// TIA Portal V19 export
FUNCTION "STD_STEP_CONTROL_HEAT" : Void   // FC6, STL
TITLE = Step controller - Heater
{ S7_Optimized_Access := 'TRUE' }
AUTHOR : JOM
FAMILY : STD
NAME : REG0391
VERSION : 0.0
// Comment
// stored: AutoNumber false
   VAR_IN_OUT
      MANUEL : Bool;   // Controller in manuel mode
      AUTO : Bool;   // Controller in auto mode
      PV : Real;   // Process Variabel
      SP : Real;   // Set Point
      MAX_DELTA : Real;
      MIN_DELTA : Real;
      FAKTOR_LARGE : Int;
      FAKTOR_SMALL : Int;
      ANA_OUTPUT : Int;
   END_VAR
BEGIN

NETWORK
TITLE = Step controller - Heater
// Comment
      A     #MANUEL;
      JC    M001;  // MANUAL
      A     #AUTO;
      JC    M002;  // AUTOMATIC
      L     0;  // = 4,00 mA
      T     #ANA_OUTPUT;  // OUTPUT
      BEU;  // END
M002: NOP   0;
      L     #PV;  // MEASURED
      L     #SP;  // SETPOINT
      -R;
      L     #MAX_DELTA;  // MAX. DELTA
      >R;
      JC    M004;
      L     #SP;  // SETPOINT
      L     #PV;  // MEASURED
      -R;
      L     #MAX_DELTA;  // MAX. DELTA
      >R;
      JC    M003;
      L     #PV;  // MEASURED
      L     #SP;  // SETPOINT
      -R;
      L     #MIN_DELTA;  // MIN. DELTA
      >R;
      JC    M006;
      L     #SP;  // SETPOINT
      L     #PV;  // MEASURED
      -R;
      L     #MIN_DELTA;  // MIN. DELTA
      >R;
      JC    M005;

      L     5000;  // IF PROCESS VALUE IS INSIDE RANGES
      T     #ANA_OUTPUT;  // THEN SET 12.00mA/5000 TO ANALOG OUTPUT

      JU    M001;
M003: L     #ANA_OUTPUT;  // OUTPUT
      L     #FAKTOR_LARGE;  // FAKTOR LARGE
      +I;
      T     #ANA_OUTPUT;  // OUTPUT
      JU    M001;
M004: L     #ANA_OUTPUT;  // OUTPUT
      L     #FAKTOR_LARGE;  // FAKTOR LARGE
      -I;
      T     #ANA_OUTPUT;  // OUTPUT
      JU    M001;
M005: L     #ANA_OUTPUT;  // OUTPUT
      L     #FAKTOR_SMALL;  // FAKTOR SMALL
      +I;
      T     #ANA_OUTPUT;  // OUTPUT
      JU    M001;
M006: L     #ANA_OUTPUT;  // OUTPUT
      L     #FAKTOR_SMALL;  // FAKTOR SMALL
      -I;
      T     #ANA_OUTPUT;  // OUTPUT
M001: L     #ANA_OUTPUT;
      L     10000;  // 20.00 mA /10000
      >I;  // > 20,00 mA
      JC    Y001;
      L     #ANA_OUTPUT;
      L     0;  // 4.00 mA / 0
      <I;  // < 4,00 mA
      JC    Y002;
      BEU;
Y001: L     10000;  // 20.00 mA / 10000
      T     #ANA_OUTPUT;
      BEU;  // = 20,00 mA
Y002: L     0;  // 4.00 mA /0
      T     #ANA_OUTPUT;
      BEU;  // = 4,00 mA
END_FUNCTION
